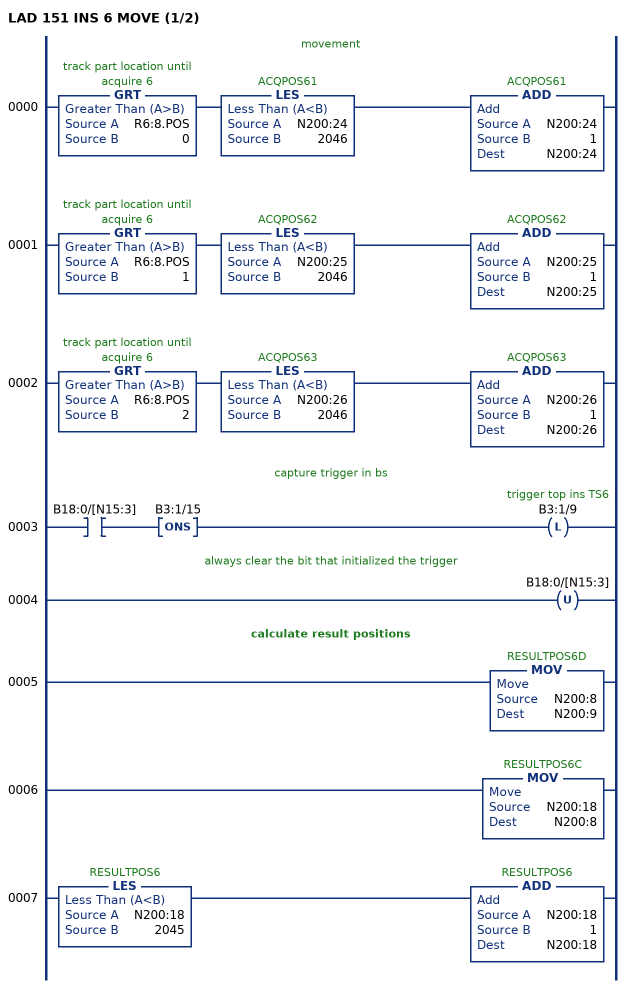
% Rung: 0 %
% movement %
SOR GRT R6:8.POS 0 LES N200:24 2046 ADD N200:24 1 N200:24 EOR
%   R6:8  "track part location until acquire 6" %
%   N200:24  ACQPOS61 %
% Rung: 1 %
SOR GRT R6:8.POS 1 LES N200:25 2046 ADD N200:25 1 N200:25 EOR
%   R6:8  "track part location until acquire 6" %
%   N200:25  ACQPOS62 %
% Rung: 2 %
SOR GRT R6:8.POS 2 LES N200:26 2046 ADD N200:26 1 N200:26 EOR
%   R6:8  "track part location until acquire 6" %
%   N200:26  ACQPOS63 %
% Rung: 3 %
% capture trigger in bs %
SOR XIC B18:0/[N15:3] ONS B3:1/15 OTL B3:1/9 EOR
%   N15:3  INS_6_TRIG_LOC %
%   B3:1/9  TS6  "trigger top ins" %
% Rung: 4 %
% always clear the bit that initialized the trigger %
SOR OTU B18:0/[N15:3] EOR
%   N15:3  INS_6_TRIG_LOC %
% Rung: 5 %
% TITLE: calculate result positions %
SOR MOV N200:8 N200:9 EOR
%   N200:8  RESULTPOS6C %
%   N200:9  RESULTPOS6D %
% Rung: 6 %
SOR MOV N200:18 N200:8 EOR
%   N200:18  RESULTPOS6 %
%   N200:8  RESULTPOS6C %
% Rung: 7 %
SOR LES N200:18 2045 ADD N200:18 1 N200:18 EOR
%   N200:18  RESULTPOS6 %

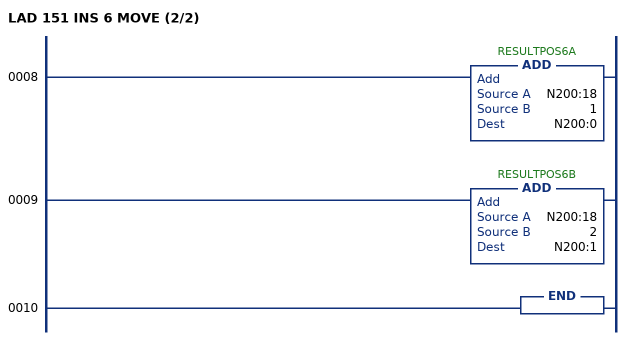
% Rung: 8 %
SOR ADD N200:18 1 N200:0 EOR
%   N200:18  RESULTPOS6 %
%   N200:0  RESULTPOS6A %
% Rung: 9 %
SOR ADD N200:18 2 N200:1 EOR
%   N200:18  RESULTPOS6 %
%   N200:1  RESULTPOS6B %
% Rung: 10 %
SOR END EOR

LADDER 160 "INS 5 TIME"
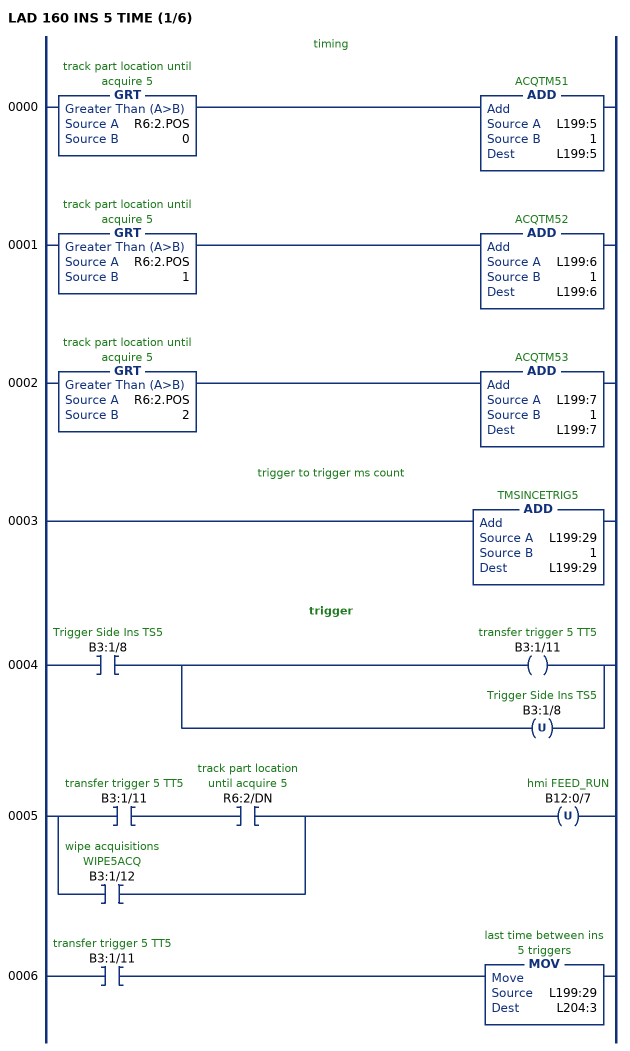
% Rung: 0 %
% timing %
SOR GRT R6:2.POS 0 ADD L199:5 1 L199:5 EOR
%   R6:2  "track part location until acquire 5" %
%   L199:5  ACQTM51 %
% Rung: 1 %
SOR GRT R6:2.POS 1 ADD L199:6 1 L199:6 EOR
%   R6:2  "track part location until acquire 5" %
%   L199:6  ACQTM52 %
% Rung: 2 %
SOR GRT R6:2.POS 2 ADD L199:7 1 L199:7 EOR
%   R6:2  "track part location until acquire 5" %
%   L199:7  ACQTM53 %
% Rung: 3 %
% trigger to trigger ms count %
SOR ADD L199:29 1 L199:29 EOR
%   L199:29  TMSINCETRIG5 %
% Rung: 4 %
% TITLE: trigger %
SOR XIC B3:1/8 BST OTE B3:1/11 NXB OTU B3:1/8 BND EOR
%   B3:1/8  TS5  "Trigger Side Ins" %
%   B3:1/11  TT5  "transfer trigger 5" %
% Rung: 5 %
SOR BST XIC B3:1/11 XIC R6:2/DN NXB XIC B3:1/12 BND OTU B12:0/7 EOR
%   B3:1/11  TT5  "transfer trigger 5" %
%   R6:2  "track part location until acquire 5" %
%   B3:1/12  WIPE5ACQ  "wipe acquisitions" %
%   B12:0/7  FEED_RUN  "hmi" %
% Rung: 6 %
SOR XIC B3:1/11 MOV L199:29 L204:3 EOR
%   B3:1/11  TT5  "transfer trigger 5" %
%   L199:29  TMSINCETRIG5 %
%   L204:3  "last time between ins 5 triggers" %

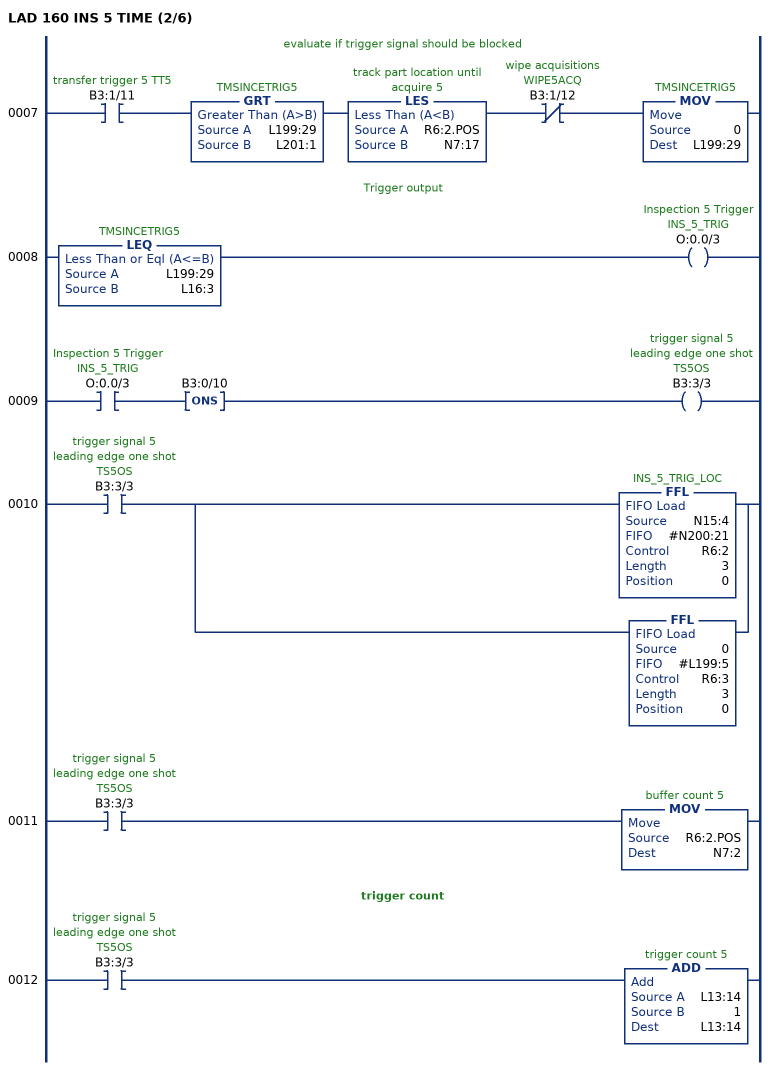
% Rung: 7 %
% evaluate if trigger signal should be blocked %
SOR XIC B3:1/11 GRT L199:29 L201:1 LES R6:2.POS N7:17 XIO B3:1/12 MOV 0 L199:29 EOR
%   B3:1/11  TT5  "transfer trigger 5" %
%   L199:29  TMSINCETRIG5 %
%   L201:1  CAM_5_MIN_CY %
%   R6:2  "track part location until acquire 5" %
%   B3:1/12  WIPE5ACQ  "wipe acquisitions" %
% Rung: 8 %
% Trigger output %
SOR LEQ L199:29 L16:3 OTE O:0.0/3 EOR
%   L199:29  TMSINCETRIG5 %
%   L16:3  CAM_5_TRIG_TIME %
%   O:0.0/3  INS_5_TRIG  "Inspection 5 Trigger" %
% Rung: 9 %
SOR XIC O:0.0/3 ONS B3:0/10 OTE B3:3/3 EOR
%   O:0.0/3  INS_5_TRIG  "Inspection 5 Trigger" %
%   B3:3/3  TS5OS  "trigger signal 5 leading edge one shot" %
% Rung: 10 %
SOR XIC B3:3/3 BST FFL N15:4 #N200:21 R6:2 3 0 NXB FFL 0 #L199:5 R6:3 3 0 BND EOR
%   B3:3/3  TS5OS  "trigger signal 5 leading edge one shot" %
%   N15:4  INS_5_TRIG_LOC %
%   N200:21  ACQPOS51 %
%   R6:2  "track part location until acquire 5" %
%   L199:5  ACQTM51 %
%   R6:3  "track acquire time 5" %
% Rung: 11 %
SOR XIC B3:3/3 MOV R6:2.POS N7:2 EOR
%   B3:3/3  TS5OS  "trigger signal 5 leading edge one shot" %
%   R6:2  "track part location until acquire 5" %
%   N7:2  "buffer count 5" %
% Rung: 12 %
% TITLE: trigger count %
SOR XIC B3:3/3 ADD L13:14 1 L13:14 EOR
%   B3:3/3  TS5OS  "trigger signal 5 leading edge one shot" %
%   L13:14  "trigger count 5" %

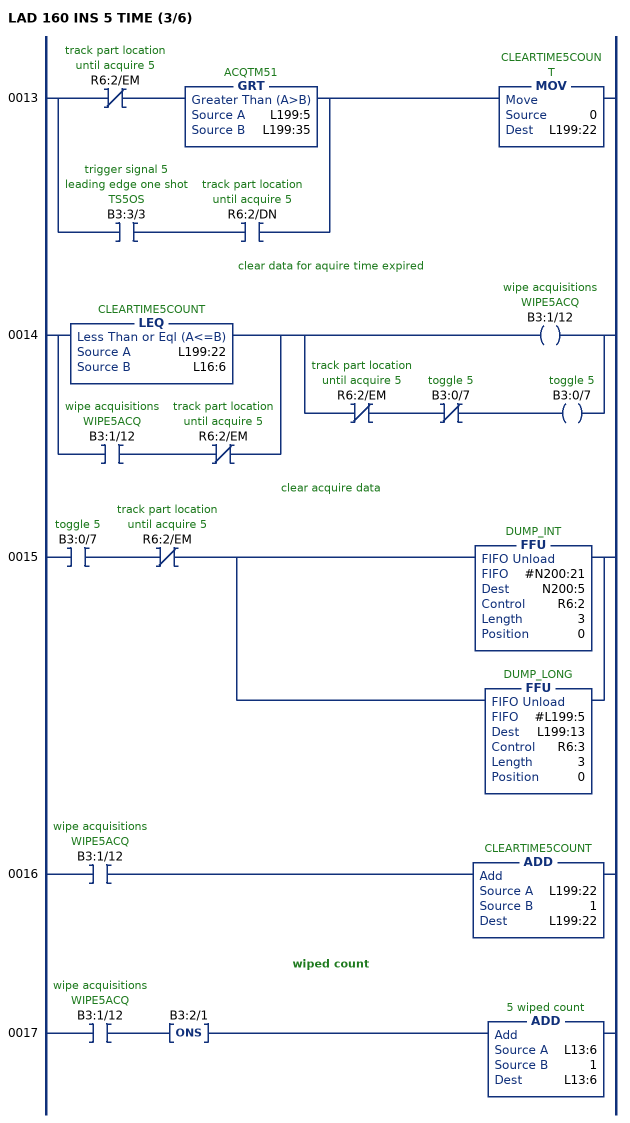
% Rung: 13 %
SOR BST XIO R6:2/EM GRT L199:5 L199:35 NXB XIC B3:3/3 XIC R6:2/DN BND MOV 0 L199:22 EOR
%   R6:2  "track part location until acquire 5" %
%   L199:5  ACQTM51 %
%   L199:35  MAXACQTM5 %
%   B3:3/3  TS5OS  "trigger signal 5 leading edge one shot" %
%   L199:22  CLEARTIME5COUNT %
% Rung: 14 %
% clear data for aquire time expired %
SOR BST LEQ L199:22 L16:6 NXB XIC B3:1/12 XIO R6:2/EM BND BST OTE B3:1/12 NXB XIO R6:2/EM XIO B3:0/7 OTE B3:0/7 BND EOR
%   L199:22  CLEARTIME5COUNT %
%   L16:6  CLEARTIME5 %
%   B3:1/12  WIPE5ACQ  "wipe acquisitions" %
%   R6:2  "track part location until acquire 5" %
%   B3:0/7  "toggle 5" %
% Rung: 15 %
% clear acquire data %
SOR XIC B3:0/7 XIO R6:2/EM BST FFU #N200:21 N200:5 R6:2 3 0 NXB FFU #L199:5 L199:13 R6:3 3 0 BND EOR
%   B3:0/7  "toggle 5" %
%   R6:2  "track part location until acquire 5" %
%   N200:21  ACQPOS51 %
%   N200:5  DUMP_INT %
%   L199:5  ACQTM51 %
%   L199:13  DUMP_LONG %
%   R6:3  "track acquire time 5" %
% Rung: 16 %
SOR XIC B3:1/12 ADD L199:22 1 L199:22 EOR
%   B3:1/12  WIPE5ACQ  "wipe acquisitions" %
%   L199:22  CLEARTIME5COUNT %
% Rung: 17 %
% TITLE: wiped count %
SOR XIC B3:1/12 ONS B3:2/1 ADD L13:6 1 L13:6 EOR
%   B3:1/12  WIPE5ACQ  "wipe acquisitions" %
%   L13:6  "5 wiped count" %

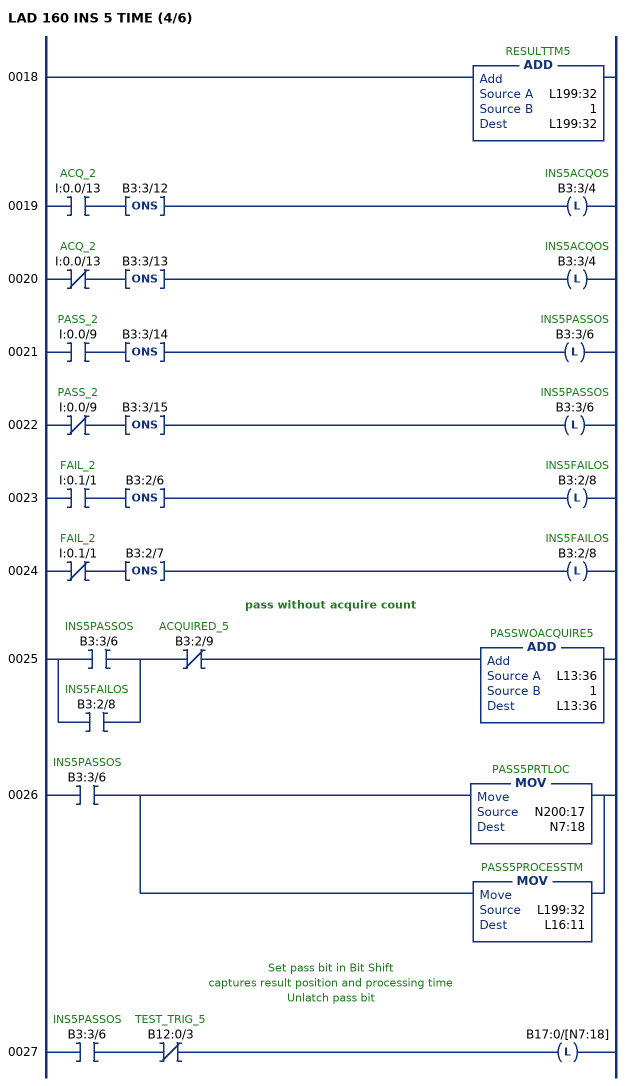
% Rung: 18 %
SOR ADD L199:32 1 L199:32 EOR
%   L199:32  RESULTTM5 %
% Rung: 19 %
SOR XIC I:0.0/13 ONS B3:3/12 OTL B3:3/4 EOR
%   I:0.0/13  ACQ_2 %
%   B3:3/4  INS5ACQOS %
% Rung: 20 %
SOR XIO I:0.0/13 ONS B3:3/13 OTL B3:3/4 EOR
%   I:0.0/13  ACQ_2 %
%   B3:3/4  INS5ACQOS %
% Rung: 21 %
SOR XIC I:0.0/9 ONS B3:3/14 OTL B3:3/6 EOR
%   I:0.0/9  PASS_2 %
%   B3:3/6  INS5PASSOS %
% Rung: 22 %
SOR XIO I:0.0/9 ONS B3:3/15 OTL B3:3/6 EOR
%   I:0.0/9  PASS_2 %
%   B3:3/6  INS5PASSOS %
% Rung: 23 %
SOR XIC I:0.1/1 ONS B3:2/6 OTL B3:2/8 EOR
%   I:0.1/1  FAIL_2 %
%   B3:2/8  INS5FAILOS %
% Rung: 24 %
SOR XIO I:0.1/1 ONS B3:2/7 OTL B3:2/8 EOR
%   I:0.1/1  FAIL_2 %
%   B3:2/8  INS5FAILOS %
% Rung: 25 %
% TITLE: pass without acquire count %
SOR BST XIC B3:3/6 NXB XIC B3:2/8 BND XIO B3:2/9 ADD L13:36 1 L13:36 EOR
%   B3:3/6  INS5PASSOS %
%   B3:2/8  INS5FAILOS %
%   B3:2/9  ACQUIRED_5 %
%   L13:36  PASSWOACQUIRE5 %
% Rung: 26 %
SOR XIC B3:3/6 BST MOV N200:17 N7:18 NXB MOV L199:32 L16:11 BND EOR
%   B3:3/6  INS5PASSOS %
%   N200:17  RESULTPOS5 %
%   N7:18  PASS5PRTLOC %
%   L199:32  RESULTTM5 %
%   L16:11  PASS5PROCESSTM %
% Rung: 27 %
% Set pass bit in Bit Shift
% captures result position and processing time
% Unlatch pass bit %
SOR XIC B3:3/6 XIO B12:0/3 OTL B17:0/[N7:18] EOR
%   B3:3/6  INS5PASSOS %
%   B12:0/3  TEST_TRIG_5 %
%   N7:18  PASS5PRTLOC %

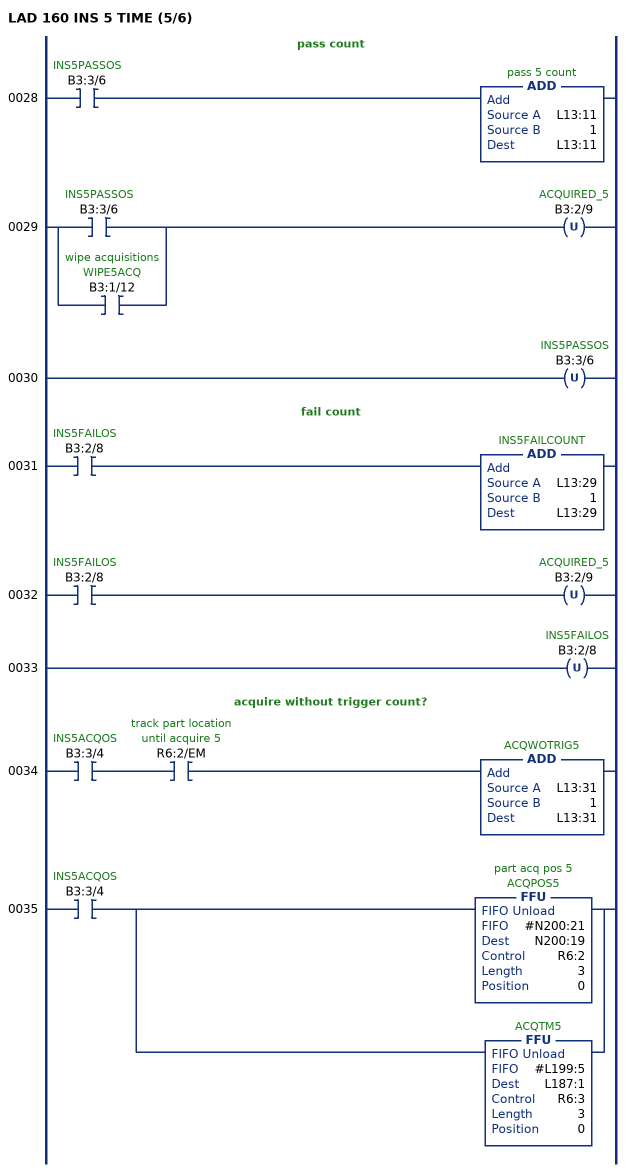
% Rung: 28 %
% TITLE: pass count %
SOR XIC B3:3/6 ADD L13:11 1 L13:11 EOR
%   B3:3/6  INS5PASSOS %
%   L13:11  "pass 5 count" %
% Rung: 29 %
SOR BST XIC B3:3/6 NXB XIC B3:1/12 BND OTU B3:2/9 EOR
%   B3:3/6  INS5PASSOS %
%   B3:1/12  WIPE5ACQ  "wipe acquisitions" %
%   B3:2/9  ACQUIRED_5 %
% Rung: 30 %
SOR OTU B3:3/6 EOR
%   B3:3/6  INS5PASSOS %
% Rung: 31 %
% TITLE: fail count %
SOR XIC B3:2/8 ADD L13:29 1 L13:29 EOR
%   B3:2/8  INS5FAILOS %
%   L13:29  INS5FAILCOUNT %
% Rung: 32 %
SOR XIC B3:2/8 OTU B3:2/9 EOR
%   B3:2/8  INS5FAILOS %
%   B3:2/9  ACQUIRED_5 %
% Rung: 33 %
SOR OTU B3:2/8 EOR
%   B3:2/8  INS5FAILOS %
% Rung: 34 %
% TITLE: acquire without trigger count? %
SOR XIC B3:3/4 XIC R6:2/EM ADD L13:31 1 L13:31 EOR
%   B3:3/4  INS5ACQOS %
%   R6:2  "track part location until acquire 5" %
%   L13:31  ACQWOTRIG5 %
% Rung: 35 %
SOR XIC B3:3/4 BST FFU #N200:21 N200:19 R6:2 3 0 NXB FFU #L199:5 L187:1 R6:3 3 0 BND EOR
%   B3:3/4  INS5ACQOS %
%   N200:21  ACQPOS51 %
%   N200:19  ACQPOS5  "part acq pos 5" %
%   R6:2  "track part location until acquire 5" %
%   L199:5  ACQTM51 %
%   L187:1  ACQTM5 %
%   R6:3  "track acquire time 5" %

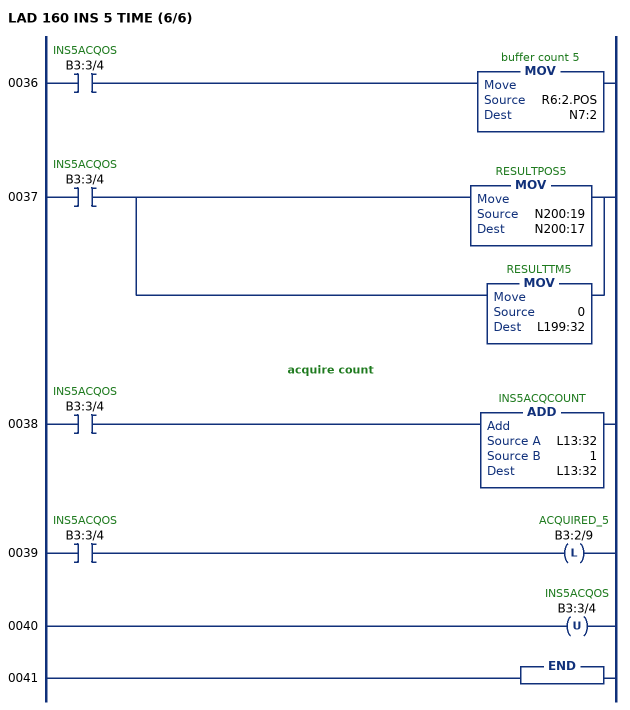
% Rung: 36 %
SOR XIC B3:3/4 MOV R6:2.POS N7:2 EOR
%   B3:3/4  INS5ACQOS %
%   R6:2  "track part location until acquire 5" %
%   N7:2  "buffer count 5" %
% Rung: 37 %
SOR XIC B3:3/4 BST MOV N200:19 N200:17 NXB MOV 0 L199:32 BND EOR
%   B3:3/4  INS5ACQOS %
%   N200:19  ACQPOS5  "part acq pos 5" %
%   N200:17  RESULTPOS5 %
%   L199:32  RESULTTM5 %
% Rung: 38 %
% TITLE: acquire count %
SOR XIC B3:3/4 ADD L13:32 1 L13:32 EOR
%   B3:3/4  INS5ACQOS %
%   L13:32  INS5ACQCOUNT %
% Rung: 39 %
SOR XIC B3:3/4 OTL B3:2/9 EOR
%   B3:3/4  INS5ACQOS %
%   B3:2/9  ACQUIRED_5 %
% Rung: 40 %
SOR OTU B3:3/4 EOR
%   B3:3/4  INS5ACQOS %
% Rung: 41 %
SOR END EOR

LADDER 161 "INS 6 TIME"
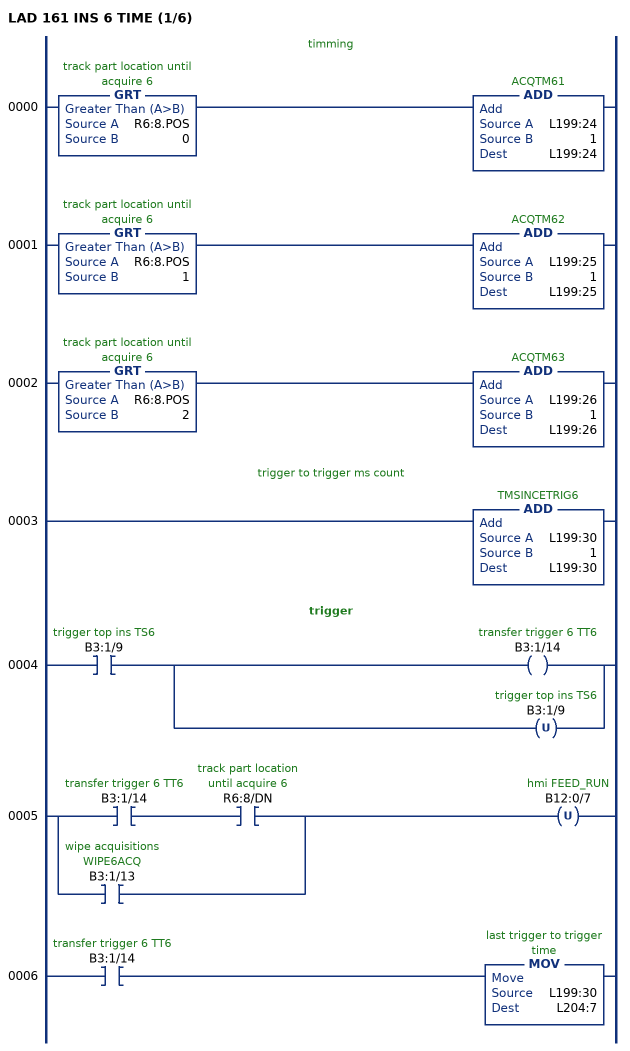
% Rung: 0 %
% timming %
SOR GRT R6:8.POS 0 ADD L199:24 1 L199:24 EOR
%   R6:8  "track part location until acquire 6" %
%   L199:24  ACQTM61 %
% Rung: 1 %
SOR GRT R6:8.POS 1 ADD L199:25 1 L199:25 EOR
%   R6:8  "track part location until acquire 6" %
%   L199:25  ACQTM62 %
% Rung: 2 %
SOR GRT R6:8.POS 2 ADD L199:26 1 L199:26 EOR
%   R6:8  "track part location until acquire 6" %
%   L199:26  ACQTM63 %
% Rung: 3 %
% trigger to trigger ms count %
SOR ADD L199:30 1 L199:30 EOR
%   L199:30  TMSINCETRIG6 %
% Rung: 4 %
% TITLE: trigger %
SOR XIC B3:1/9 BST OTE B3:1/14 NXB OTU B3:1/9 BND EOR
%   B3:1/9  TS6  "trigger top ins" %
%   B3:1/14  TT6  "transfer trigger 6" %
% Rung: 5 %
SOR BST XIC B3:1/14 XIC R6:8/DN NXB XIC B3:1/13 BND OTU B12:0/7 EOR
%   B3:1/14  TT6  "transfer trigger 6" %
%   R6:8  "track part location until acquire 6" %
%   B3:1/13  WIPE6ACQ  "wipe acquisitions" %
%   B12:0/7  FEED_RUN  "hmi" %
% Rung: 6 %
SOR XIC B3:1/14 MOV L199:30 L204:7 EOR
%   B3:1/14  TT6  "transfer trigger 6" %
%   L199:30  TMSINCETRIG6 %
%   L204:7  "last trigger to trigger time" %

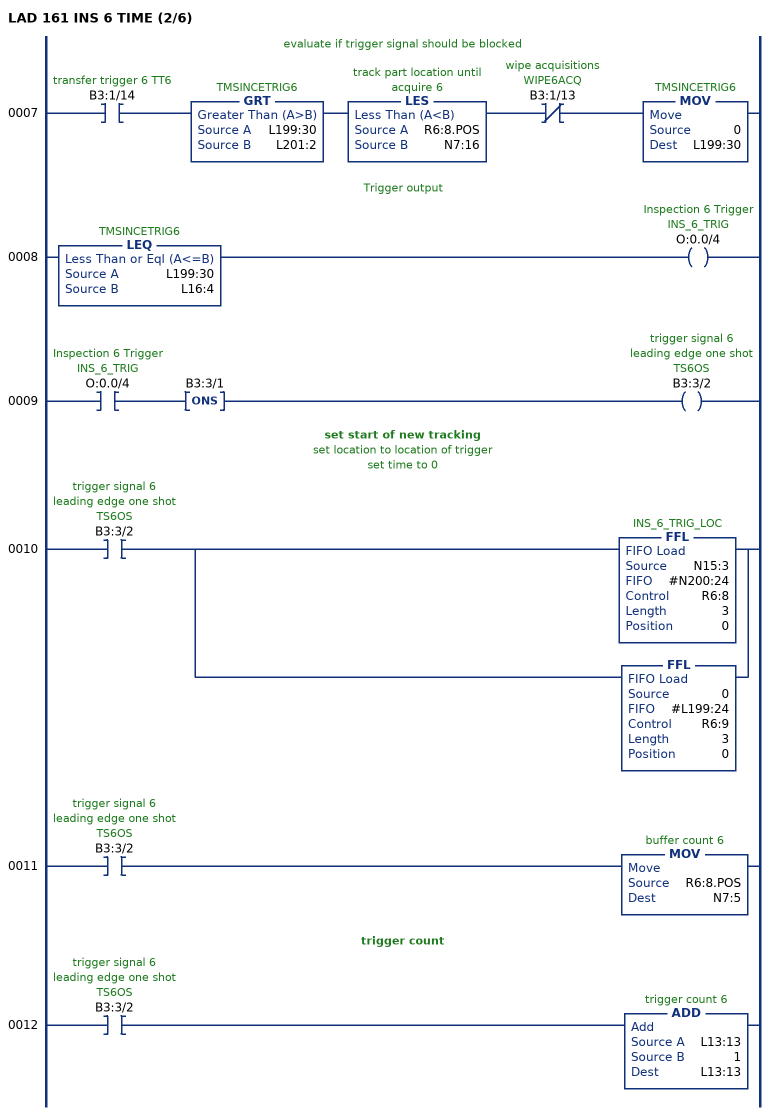
% Rung: 7 %
% evaluate if trigger signal should be blocked %
SOR XIC B3:1/14 GRT L199:30 L201:2 LES R6:8.POS N7:16 XIO B3:1/13 MOV 0 L199:30 EOR
%   B3:1/14  TT6  "transfer trigger 6" %
%   L199:30  TMSINCETRIG6 %
%   L201:2  CAM_6_MIN_CY %
%   R6:8  "track part location until acquire 6" %
%   B3:1/13  WIPE6ACQ  "wipe acquisitions" %
% Rung: 8 %
% Trigger output %
SOR LEQ L199:30 L16:4 OTE O:0.0/4 EOR
%   L199:30  TMSINCETRIG6 %
%   L16:4  CAM_6_TRIG_TIME %
%   O:0.0/4  INS_6_TRIG  "Inspection 6 Trigger" %
% Rung: 9 %
SOR XIC O:0.0/4 ONS B3:3/1 OTE B3:3/2 EOR
%   O:0.0/4  INS_6_TRIG  "Inspection 6 Trigger" %
%   B3:3/2  TS6OS  "trigger signal 6 leading edge one shot" %
% Rung: 10 %
% TITLE: set start of new tracking %
% set location to location of trigger
% set time to 0 %
SOR XIC B3:3/2 BST FFL N15:3 #N200:24 R6:8 3 0 NXB FFL 0 #L199:24 R6:9 3 0 BND EOR
%   B3:3/2  TS6OS  "trigger signal 6 leading edge one shot" %
%   N15:3  INS_6_TRIG_LOC %
%   N200:24  ACQPOS61 %
%   R6:8  "track part location until acquire 6" %
%   L199:24  ACQTM61 %
%   R6:9  "track acquire time 6" %
% Rung: 11 %
SOR XIC B3:3/2 MOV R6:8.POS N7:5 EOR
%   B3:3/2  TS6OS  "trigger signal 6 leading edge one shot" %
%   R6:8  "track part location until acquire 6" %
%   N7:5  "buffer count 6" %
% Rung: 12 %
% TITLE: trigger count %
SOR XIC B3:3/2 ADD L13:13 1 L13:13 EOR
%   B3:3/2  TS6OS  "trigger signal 6 leading edge one shot" %
%   L13:13  "trigger count 6" %

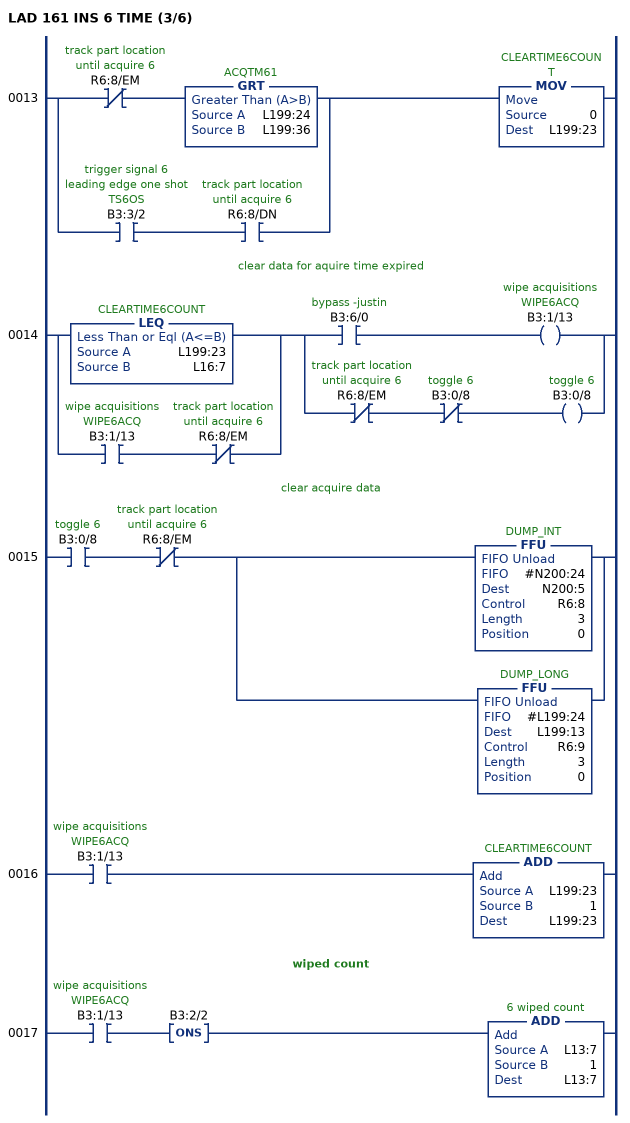
% Rung: 13 %
SOR BST XIO R6:8/EM GRT L199:24 L199:36 NXB XIC B3:3/2 XIC R6:8/DN BND MOV 0 L199:23 EOR
%   R6:8  "track part location until acquire 6" %
%   L199:24  ACQTM61 %
%   L199:36  MAXACQTM6 %
%   B3:3/2  TS6OS  "trigger signal 6 leading edge one shot" %
%   L199:23  CLEARTIME6COUNT %
% Rung: 14 %
% clear data for aquire time expired %
SOR BST LEQ L199:23 L16:7 NXB XIC B3:1/13 XIO R6:8/EM BND BST XIC B3:6/0 OTE B3:1/13 NXB XIO R6:8/EM XIO B3:0/8 OTE B3:0/8 BND EOR
%   L199:23  CLEARTIME6COUNT %
%   L16:7  CLEARTIME6 %
%   B3:1/13  WIPE6ACQ  "wipe acquisitions" %
%   R6:8  "track part location until acquire 6" %
%   B3:6/0  "bypass -justin" %
%   B3:0/8  "toggle 6" %
% Rung: 15 %
% clear acquire data %
SOR XIC B3:0/8 XIO R6:8/EM BST FFU #N200:24 N200:5 R6:8 3 0 NXB FFU #L199:24 L199:13 R6:9 3 0 BND EOR
%   B3:0/8  "toggle 6" %
%   R6:8  "track part location until acquire 6" %
%   N200:24  ACQPOS61 %
%   N200:5  DUMP_INT %
%   L199:24  ACQTM61 %
%   L199:13  DUMP_LONG %
%   R6:9  "track acquire time 6" %
% Rung: 16 %
SOR XIC B3:1/13 ADD L199:23 1 L199:23 EOR
%   B3:1/13  WIPE6ACQ  "wipe acquisitions" %
%   L199:23  CLEARTIME6COUNT %
% Rung: 17 %
% TITLE: wiped count %
SOR XIC B3:1/13 ONS B3:2/2 ADD L13:7 1 L13:7 EOR
%   B3:1/13  WIPE6ACQ  "wipe acquisitions" %
%   L13:7  "6 wiped count" %

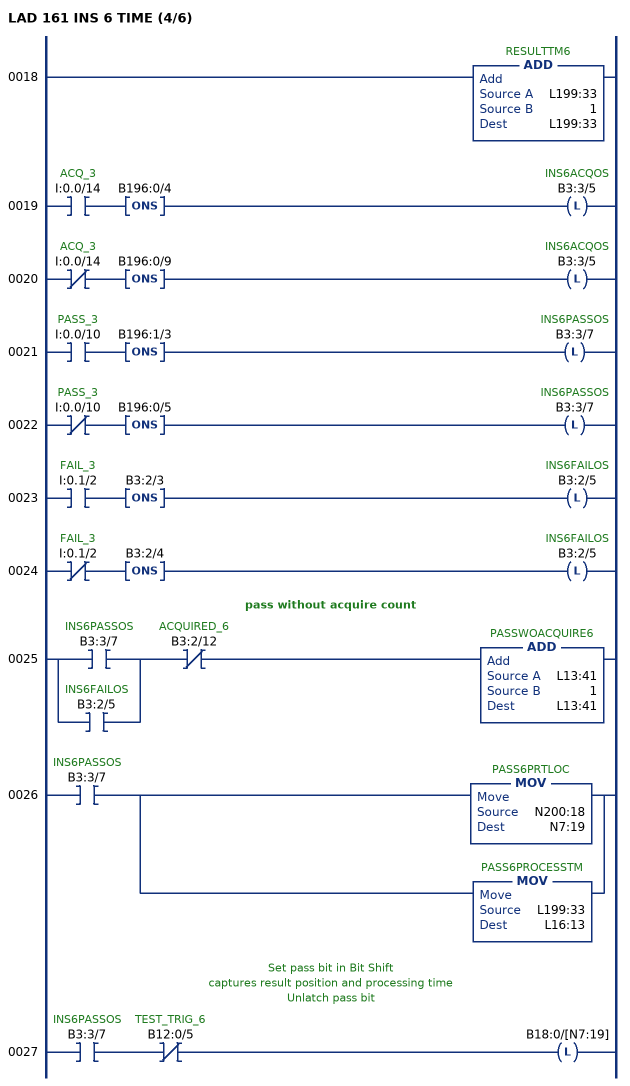
% Rung: 18 %
SOR ADD L199:33 1 L199:33 EOR
%   L199:33  RESULTTM6 %
% Rung: 19 %
SOR XIC I:0.0/14 ONS B196:0/4 OTL B3:3/5 EOR
%   I:0.0/14  ACQ_3 %
%   B3:3/5  INS6ACQOS %
% Rung: 20 %
SOR XIO I:0.0/14 ONS B196:0/9 OTL B3:3/5 EOR
%   I:0.0/14  ACQ_3 %
%   B3:3/5  INS6ACQOS %
% Rung: 21 %
SOR XIC I:0.0/10 ONS B196:1/3 OTL B3:3/7 EOR
%   I:0.0/10  PASS_3 %
%   B3:3/7  INS6PASSOS %
% Rung: 22 %
SOR XIO I:0.0/10 ONS B196:0/5 OTL B3:3/7 EOR
%   I:0.0/10  PASS_3 %
%   B3:3/7  INS6PASSOS %
% Rung: 23 %
SOR XIC I:0.1/2 ONS B3:2/3 OTL B3:2/5 EOR
%   I:0.1/2  FAIL_3 %
%   B3:2/5  INS6FAILOS %
% Rung: 24 %
SOR XIO I:0.1/2 ONS B3:2/4 OTL B3:2/5 EOR
%   I:0.1/2  FAIL_3 %
%   B3:2/5  INS6FAILOS %
% Rung: 25 %
% TITLE: pass without acquire count %
SOR BST XIC B3:3/7 NXB XIC B3:2/5 BND XIO B3:2/12 ADD L13:41 1 L13:41 EOR
%   B3:3/7  INS6PASSOS %
%   B3:2/5  INS6FAILOS %
%   B3:2/12  ACQUIRED_6 %
%   L13:41  PASSWOACQUIRE6 %
% Rung: 26 %
SOR XIC B3:3/7 BST MOV N200:18 N7:19 NXB MOV L199:33 L16:13 BND EOR
%   B3:3/7  INS6PASSOS %
%   N200:18  RESULTPOS6 %
%   N7:19  PASS6PRTLOC %
%   L199:33  RESULTTM6 %
%   L16:13  PASS6PROCESSTM %
% Rung: 27 %
% Set pass bit in Bit Shift
% captures result position and processing time
% Unlatch pass bit %
SOR XIC B3:3/7 XIO B12:0/5 OTL B18:0/[N7:19] EOR
%   B3:3/7  INS6PASSOS %
%   B12:0/5  TEST_TRIG_6 %
%   N7:19  PASS6PRTLOC %

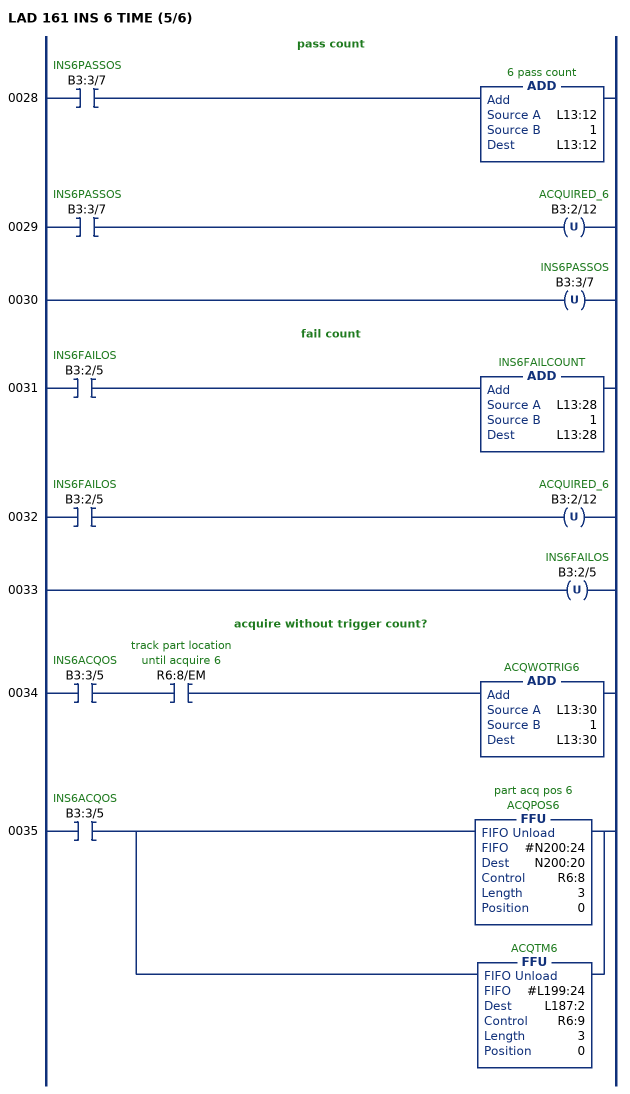
% Rung: 28 %
% TITLE: pass count %
SOR XIC B3:3/7 ADD L13:12 1 L13:12 EOR
%   B3:3/7  INS6PASSOS %
%   L13:12  "6 pass count" %
% Rung: 29 %
SOR XIC B3:3/7 OTU B3:2/12 EOR
%   B3:3/7  INS6PASSOS %
%   B3:2/12  ACQUIRED_6 %
% Rung: 30 %
SOR OTU B3:3/7 EOR
%   B3:3/7  INS6PASSOS %
% Rung: 31 %
% TITLE: fail count %
SOR XIC B3:2/5 ADD L13:28 1 L13:28 EOR
%   B3:2/5  INS6FAILOS %
%   L13:28  INS6FAILCOUNT %
% Rung: 32 %
SOR XIC B3:2/5 OTU B3:2/12 EOR
%   B3:2/5  INS6FAILOS %
%   B3:2/12  ACQUIRED_6 %
% Rung: 33 %
SOR OTU B3:2/5 EOR
%   B3:2/5  INS6FAILOS %
% Rung: 34 %
% TITLE: acquire without trigger count? %
SOR XIC B3:3/5 XIC R6:8/EM ADD L13:30 1 L13:30 EOR
%   B3:3/5  INS6ACQOS %
%   R6:8  "track part location until acquire 6" %
%   L13:30  ACQWOTRIG6 %
% Rung: 35 %
SOR XIC B3:3/5 BST FFU #N200:24 N200:20 R6:8 3 0 NXB FFU #L199:24 L187:2 R6:9 3 0 BND EOR
%   B3:3/5  INS6ACQOS %
%   N200:24  ACQPOS61 %
%   N200:20  ACQPOS6  "part acq pos 6" %
%   R6:8  "track part location until acquire 6" %
%   L199:24  ACQTM61 %
%   L187:2  ACQTM6 %
%   R6:9  "track acquire time 6" %

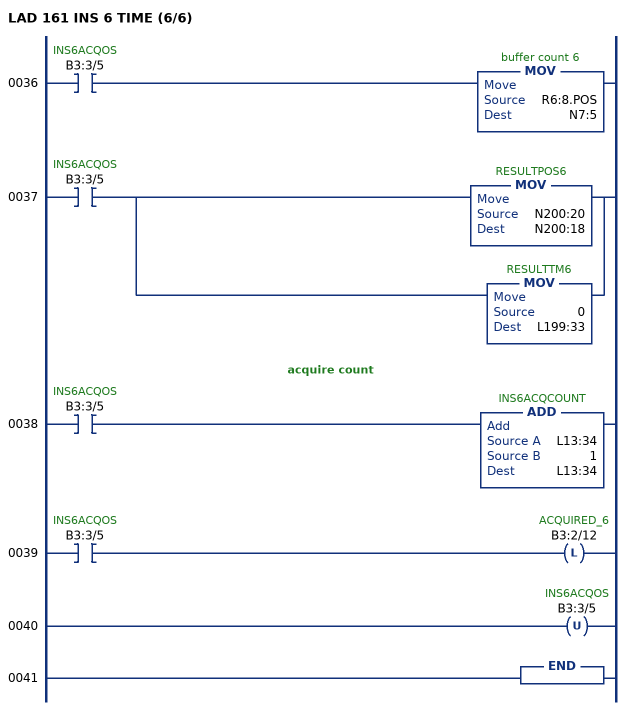
% Rung: 36 %
SOR XIC B3:3/5 MOV R6:8.POS N7:5 EOR
%   B3:3/5  INS6ACQOS %
%   R6:8  "track part location until acquire 6" %
%   N7:5  "buffer count 6" %
% Rung: 37 %
SOR XIC B3:3/5 BST MOV N200:20 N200:18 NXB MOV 0 L199:33 BND EOR
%   B3:3/5  INS6ACQOS %
%   N200:20  ACQPOS6  "part acq pos 6" %
%   N200:18  RESULTPOS6 %
%   L199:33  RESULTTM6 %
% Rung: 38 %
% TITLE: acquire count %
SOR XIC B3:3/5 ADD L13:34 1 L13:34 EOR
%   B3:3/5  INS6ACQOS %
%   L13:34  INS6ACQCOUNT %
% Rung: 39 %
SOR XIC B3:3/5 OTL B3:2/12 EOR
%   B3:3/5  INS6ACQOS %
%   B3:2/12  ACQUIRED_6 %
% Rung: 40 %
SOR OTU B3:3/5 EOR
%   B3:3/5  INS6ACQOS %
% Rung: 41 %
SOR END EOR

LADDER 170 "PASS BLOW"
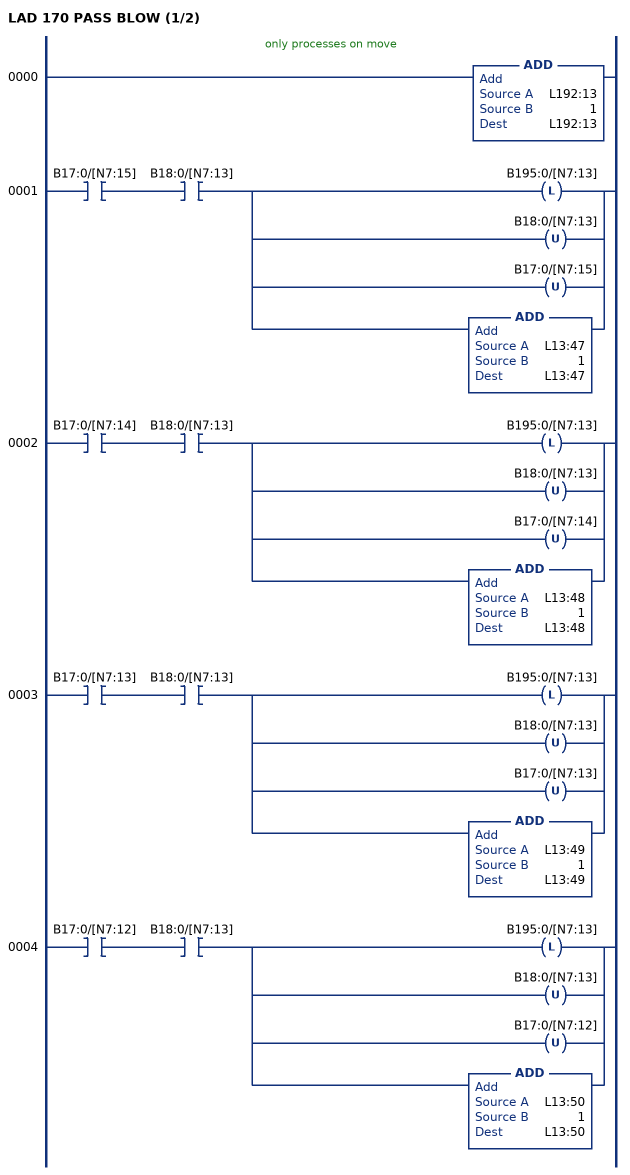
% Rung: 0 %
% only processes on move %
SOR ADD L192:13 1 L192:13 EOR
% Rung: 1 %
SOR XIC B17:0/[N7:15] XIC B18:0/[N7:13] BST OTL B195:0/[N7:13] NXB OTU B18:0/[N7:13] NXB OTU B17:0/[N7:15] NXB ADD L13:47 1 L13:47 BND EOR
%   N7:15  OS5 %
%   N7:13  OS3 %
% Rung: 2 %
SOR XIC B17:0/[N7:14] XIC B18:0/[N7:13] BST OTL B195:0/[N7:13] NXB OTU B18:0/[N7:13] NXB OTU B17:0/[N7:14] NXB ADD L13:48 1 L13:48 BND EOR
%   N7:14  OS4 %
%   N7:13  OS3 %
% Rung: 3 %
SOR XIC B17:0/[N7:13] XIC B18:0/[N7:13] BST OTL B195:0/[N7:13] NXB OTU B18:0/[N7:13] NXB OTU B17:0/[N7:13] NXB ADD L13:49 1 L13:49 BND EOR
%   N7:13  OS3 %
% Rung: 4 %
SOR XIC B17:0/[N7:12] XIC B18:0/[N7:13] BST OTL B195:0/[N7:13] NXB OTU B18:0/[N7:13] NXB OTU B17:0/[N7:12] NXB ADD L13:50 1 L13:50 BND EOR
%   N7:12  OS2 %
%   N7:13  OS3 %

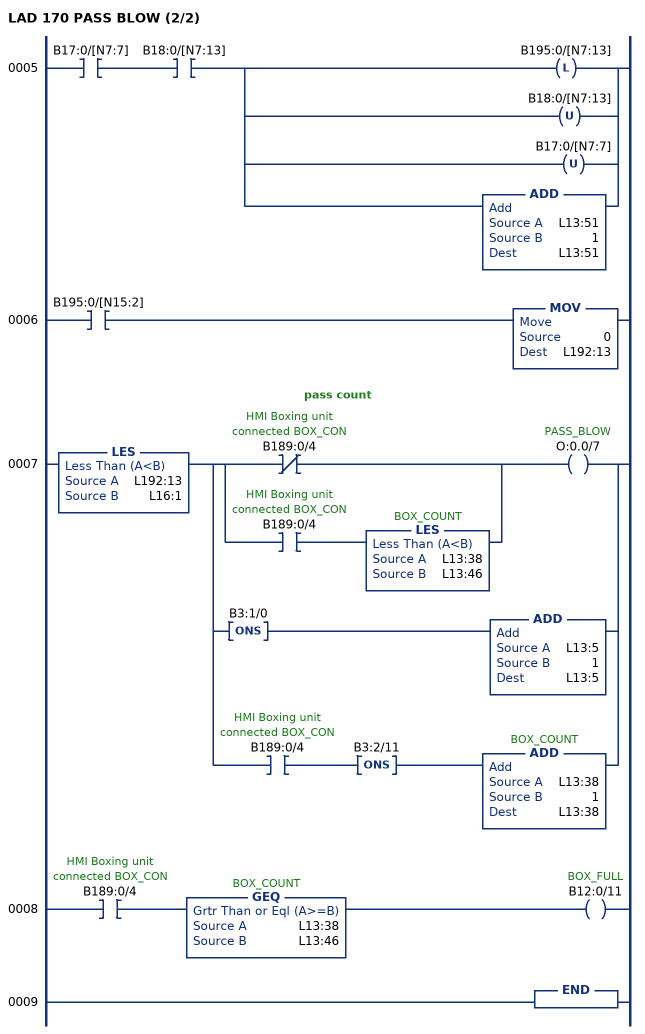
% Rung: 5 %
SOR XIC B17:0/[N7:7] XIC B18:0/[N7:13] BST OTL B195:0/[N7:13] NXB OTU B18:0/[N7:13] NXB OTU B17:0/[N7:7] NXB ADD L13:51 1 L13:51 BND EOR
%   N7:7  OS1 %
%   N7:13  OS3 %
% Rung: 6 %
SOR XIC B195:0/[N15:2] MOV 0 L192:13 EOR
%   N15:2  BLOW_PT %
% Rung: 7 %
% TITLE: pass count %
SOR LES L192:13 L16:1 BST BST XIO B189:0/4 NXB XIC B189:0/4 LES L13:38 L13:46 BND OTE O:0.0/7 NXB ONS B3:1/0 ADD L13:5 1 L13:5 NXB XIC B189:0/4 ONS B3:2/11 ADD L13:38 1 L13:38 BND EOR
%   L16:1  BLOW_TIME %
%   B189:0/4  BOX_CON  "HMI Boxing unit connected" %
%   L13:38  BOX_COUNT %
%   L13:46  BOX_LIMIT  "box count setpoint" %
%   O:0.0/7  PASS_BLOW %
% Rung: 8 %
SOR XIC B189:0/4 GEQ L13:38 L13:46 OTE B12:0/11 EOR
%   B189:0/4  BOX_CON  "HMI Boxing unit connected" %
%   L13:38  BOX_COUNT %
%   L13:46  BOX_LIMIT  "box count setpoint" %
%   B12:0/11  BOX_FULL %
% Rung: 9 %
SOR END EOR

LADDER 180 "RATE"
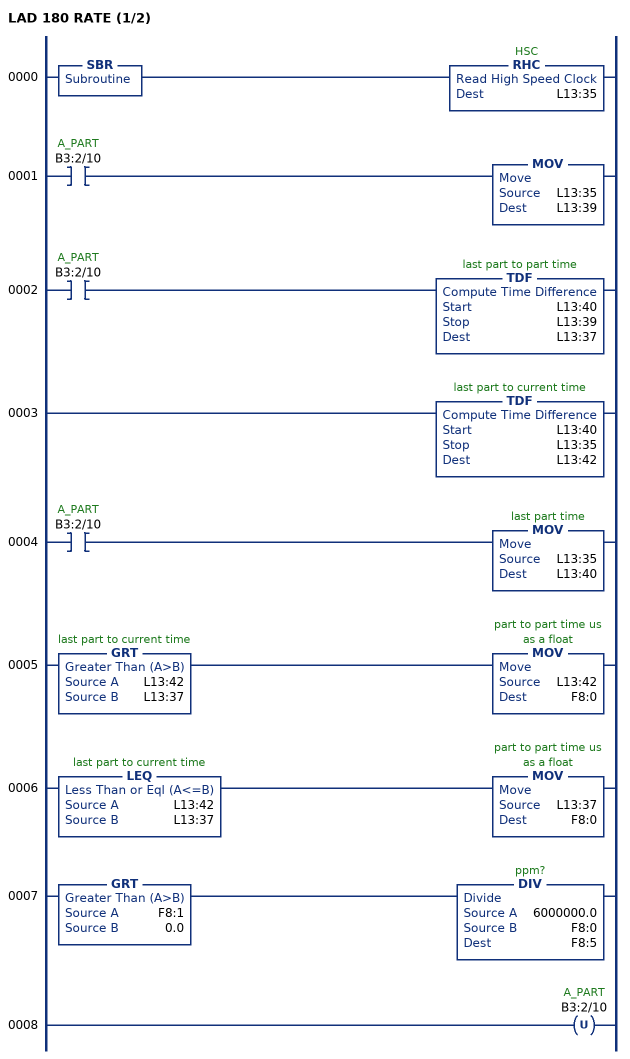
% Rung: 0 %
SOR SBR RHC L13:35 EOR
%   L13:35  HSC %
% Rung: 1 %
SOR XIC B3:2/10 MOV L13:35 L13:39 EOR
%   B3:2/10  A_PART %
%   L13:35  HSC %
% Rung: 2 %
SOR XIC B3:2/10 TDF L13:40 L13:39 L13:37 EOR
%   B3:2/10  A_PART %
%   L13:40  "last part time" %
%   L13:37  "last part to part time" %
% Rung: 3 %
SOR TDF L13:40 L13:35 L13:42 EOR
%   L13:40  "last part time" %
%   L13:35  HSC %
%   L13:42  "last part to current time" %
% Rung: 4 %
SOR XIC B3:2/10 MOV L13:35 L13:40 EOR
%   B3:2/10  A_PART %
%   L13:35  HSC %
%   L13:40  "last part time" %
% Rung: 5 %
SOR GRT L13:42 L13:37 MOV L13:42 F8:0 EOR
%   L13:42  "last part to current time" %
%   L13:37  "last part to part time" %
%   F8:0  "part to part time us as a float" %
% Rung: 6 %
SOR LEQ L13:42 L13:37 MOV L13:37 F8:0 EOR
%   L13:42  "last part to current time" %
%   L13:37  "last part to part time" %
%   F8:0  "part to part time us as a float" %
% Rung: 7 %
SOR GRT F8:1 0.0 DIV 6000000.0 F8:0 F8:5 EOR
%   F8:0  "part to part time us as a float" %
%   F8:5  "ppm?" %
% Rung: 8 %
SOR OTU B3:2/10 EOR
%   B3:2/10  A_PART %

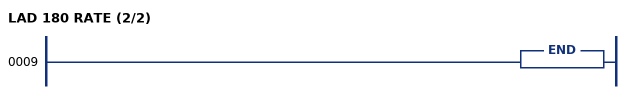
% Rung: 9 %
SOR END EOR

OTHER DOCUMENTED ADDRESSES
  B3:8/1  "bypass extra trigger camera 2"
  B3:8/2  "bypass extra trigger camera 3"
  B3:8/3  "bypass extra trigger camera 4"
  B3:8/6  "a bypass bit"
  B3:8/7  "a bypass bit"
  B3:8/12  "start bottom top camera responce"
  B3:8/13  "extra blow signal for testing"
  B3:8/15  "start side camera responce"
  B3:9/2  "one shot"
  B3:9/4  "start top camera responce"
  B3:9/6  "C1D"
  B3:9/7  "C1t"
  B3:9/8  "C2D"
  B3:9/9  "C2t"
  B3:9/14  "input from hmi to reset count"
  B3:10/0  "bypass part too close"
  B3:10/2  "One Shot"
  B3:10/3  "One Shot"
  B3:10/4  "changing Box chute door operation"
  B3:10/5  "one shot"
  B3:10/6  "excessive data output time"
  B3:10/9  "one shot"
  B3:10/10  "one shot"
  B3:10/11  "bottom part present trailling edge"
  B3:10/13  "one shot"
  B3:10/14  "Dont use"
  B3:10/15  "Reserved For Shift Registers"
  B3:11/0  "bypass unused portion of code"
  B3:11/1  "bypass"
  B3:11/2  "Enable encoder belt movement simulation when testing"
  B3:11/3  "Block blow signals while changing box"
  B3:11/4  "one shot"
  B3:11/6  "one shot"
  B3:11/7  "one shot"
  B3:11/8  "one shot"
  B3:11/11  "one shot"
  B3:11/12  "one shot"
  B3:11/15  "one shot"
  B3:12/0  "one shot"
  B3:12/1  "one shot"
  B3:12/2  "Command 2 Oneshot"
  B3:12/3  "Command 2 Active"
  B3:12/4  "Command3 Oneshot"
  B3:12/5  "Command 3 Active"
  B3:12/6  "Inspection Command Counter"
  B3:12/7  "Command 4 Active"
  B3:12/8  "Command 4 Oneshot"
  B3:12/14  "flip flop bit"
  B3:13/5  "bypass"
  B3:13/6  "Off"
  B3:13/7  "On"
  B3:13/8  "On"
  B3:13/9  "Off"
  B3:13/10  "On"
  B3:13/11  "Off"
  B3:13/12  "Test Trigger to laser Spacing"
  B3:13/15  "Test Signals"
  B3:17/12  "Always Off"
  B9:0/0  "Trigger Insert Position"
  B9:0/1  "bottom of top conveyor part transfer location"
  B9:0/[N7:0]  "Side Camera Trigger Posistion"
  B9:0/[N7:2]  "Mask Start Position"
  B9:0/[N7:6]  "Blow Off Position"
  B9:0/[N7:20]  "part present bit shift load position"
  B9:0/[N7:48]  "Top Camera Trigger Posistion"
  B9:0/[N16:0]  "Trigger Position"
  B9:0/[N17:8]  "part from bottom belt present at top belt optic position"
  B10:0/0  "Pass Insert Position"
  B10:0/[N7:2]  "Pass Bit Position"
  B10:0/[N7:4]  "Pass Insert Position"
  B10:0/[N7:5]  "Pass Start Position"
  B10:0/[N7:6]  "Pass Position"
  B10:0/[N16:4]  "Pass Insert Position"
  B10:0/[N16:6]  "Pass Position"
  B11:0/0  "Trigger Insert Position"
  B11:0/[N7:8]  "Fail Bit Position"
  B11:0/[N16:0]  "Trigger Position"
  B12:1/0  "Conveyor Start Oneshot"
  B12:1/1  "Feed Start Oneshot"
  B12:1/2  "Conveyor Stop Oneshot"
  B12:1/3  "Feed Stop Oneshot"
  B12:1/5  "Conveyor Start Oneshot"
  B12:10  BULK_PACK
  B14:0/0  "Bottom Pass Insert"
  B14:0/4  "Bottom Pass Insert Position"
  B14:0/[N13:14]  "Start Laser Pass"
  B14:0/[N16:4]  "Pass Insert Position"
  B14:0/[N16:6]  "Pass Position"
  B15:0  "Alarm Bits"
  B18:1/1  "bottom pass one shot transfer"
  B18:3/2  "Part Present Oneshot"
  B18:3/3  "Part Present Oneshot"
  B18:5/11  "Transfer bottom pass result from end of bottom conveyor"
  B18:10/15  "Reserved For Shift Registers"
  B18:142  "fack camerea pass signal"
  B22:0  "Transfer Shift Register"
  B22:0/0  "load top conveyor bitshift from bottom cammera pass."
  B22:0/[N17:8]  "bottom good part at top optic position"
  B23:0/[N7:0]  "Bottom Pass Output"
  B185:0/0  "bypass"
  B185:0/1  "bypass"
  B185:0/9  "result time 1 okay"
  B185:0/11  "test fail out"
  B185:0/12  "enable"
  B185:0/13  "enable"
  B185:1/0  "enable"
  B185:1/3  "enable"
  B185:1/7  "enable"
  B191:1/0  "Part measured wider then the limit set in the optic test"
  B191:1/1  "part to part spacing smaller then the set minimum value"
  B191:1/2  "Boxing conveyor backed up"
  B191:2/0  "bottom to top alignment"
  B196:0/13  "waiting for result"
  B196:0/14  "acquire before result os"
  B196:0/15  "enable count"
  B196:1/5  "switch me to EN_1"
  B196:1/9  "Enable alignment Signal"
  B196:1/11  "enable"
  B196:1/12  "enable"
  B196:1/15  "transfer trigger for position alignment logical one shot"
  B196:2/0  "enable"
  B196:2/2  "enable"
  B196:2/8  "enable count"
  B196:2/9  "time out 1"
  B196:2/10  "Reset bad head fault"
  B196:4/0  "test trigger signal 1"
  B196:4/4  "real part within distance of virtual part"
  B196:4/15  "pass in bit shift"
  F8:13  "error top"
  F8:15  "error bottom"
  F8:20  "bot belt speed average in pulses per second"
  F8:26  "Part bits loaded into BitShift"
  F8:28  "momentary rate in ppm"
  F8:29  "Count of signals passed to the blow valve"
  F8:31  "Count of off alignment between top and bottom ALIGN_FAILS"
  F8:34  "count of blow signals"
  F8:35  "rate difference"
  F8:38  "averaged rate"
  F8:40  "absoloute difference top"
  F8:41  "absoloute difference bottom"
  F8:42  "Total fail and missed count CAM_NON_PASS"
  F8:43  "change in part rate as %"
  F8:44  "difference as a ratio of the total"
  F8:45  "TOO_CLOSE_BOT"
  F8:46  "TOO_WIDE_BOT"
  F8:48  "transfer"
  F8:49  "TOO_CLOSE_TOP"
  F8:51  "TOO_WIDE_TOP"
  F8:52  "OPTO_FAILS"
  F8:53  "optic fail count top camera TOP_OPT_FAIL_CT"
  F8:54  "optic fail count bot camera BOT_OPT_FAIL_CT"
  F19:4  "Conveyor Input Blip Counter"
  F188:1  "HMI Recerk speed input"
  F188:2  "HMI input for feed wheel speed"
  F188:3  "HMI input for feeder speed"
  F188:4  "HMI input for hopper speed"
  F192:0  "temp"
  F205:0  "feed wheel"
  F205:1  "feed bowl"
  F205:2  "hopper"
  HSC:0.3/6  "Underflow interrupt"
  HSC:0.3/7  "Overflow interrupt"
  HSC:1.3/6  "Underflow interrupt"
  HSC:1.3/7  "Overflow interrupt"
  I:0.0/0  "Encoder Signal "A""
  I:0.0/1  "Encoder Signal "B""
  I:0.0/4  "Encoder Signal "A""
  I:0.0/5  "Encoder Signal "B""
  I:0.0/11  PASS_4
  I:0.0/15  ACQ_4
  I:0.1/3  FAIL_4
  I:0.2/3  "Packaging Conveyor full"
  I:0.2/4  "Packaging Conveyor Box in Position"
  I:0.4  "Spare Analog Input 1"
  I:0.5  "Spare Analog Input 2"
  I:0.6  "Spare Analog Input 3"
  I:2.0/1  REAR_ESTOP
  I:2.0/8  "front door signal"
  I:2.0/9  "rear door signal"
  I:2.0/10  "Maintenance Key Switch"
  I:2.0/12  "input from customer Packager Concluded"
  L23:1  MPCE_ON
  L23:19  TOP_OPT_FAIL_CT
  L23:34  AIR_PRESSURE_FAULT
  L183:2  "simulated part width"
  L187:5  "pass transfer out signals"
  L187:6  "NoErr transfer out signals"
  L187:7  "ins 1 trigger count"
  L190:0  "count of bottom optic width fails"
  L190:1  "count of gap fails"
  L190:2  "I1 blocked triggers"
  L190:4  "count of parts rejected because acquire time ran out"
  L190:5  "count of parts that received a pass signal but previously failed 1"
  L190:6  "count of result signals received with no part present 1"
  L190:7  "count of results received after maximim time reached"
  L190:8  "pass count"
  L190:9  "fail count"
  L190:10  "acquisition count"
  L190:11  "acquisition without result count"
  L190:12  "count of parts results that time out"
  L190:27  "optic alignment pass signal"
  L190:28  "optic alignment fail signal"
  L190:31  "something wrong, can't happen"
  L190:32  "Crazy wrong, can't happen"
  L201:5  "ms since trig 1 is initialized"
  L201:10  "movement from virtual (pos, add)"
  L204:13  "This optic signal time"
  L204:14  "Last optic signal time"
  L204:15  "time between optic signals"
  N10:1  "old ConveyorStatus"
  N10:2  "PowerOn"
  N10:3  "Local Mode On BypassBoxingPLC"
  N10:4  "Boxing Connected Signal"
  N10:5  "BoxJamSignal"
  N10:6  "WaittingOnBoxSig"
  N10:7  "ConveyorFullSig"
  N10:8  "MachineFaultSig"
  N10:9  "Counter Sensor Fault"
  N10:11  "Feeder Track Sensor Blocked"
  N10:12  "Air Pressure Fault"
  N13:0  "Part Inspecting"
  N13:4  "Completed Counter"
  N13:5  "Trigger Position Counter"
  N13:6  "BlowOff Start Counter"
  N13:7  "BlowOff Stop Counter"
  N13:8  "Inspection Command Counter"
  N13:9  "Complete Counter"
  N13:10  "Pass Signal Counter"
  N13:11  "Solenoid Signal Counter"
  N13:12  "Hold Pass Counter"
  N13:13  "Hold Pass Length"
  N16:1  "Bottom Inspection Offset For Tracking"
  N16:3  "Bit Shift Preset"
  N17:5  "Parts In Tube Counter"
  N17:6  "Parts In Tube Limit"
  N17:9  "Bot to Top Transfer Position"
  N17:12  "Trigger to laser Counter"
  N197:1  "maximim acquire time 1"
  N197:5  "Feeder Speed Output Setting"
  N197:10  "pulse distance to keep blow on then turn off feed"
  N197:11  "speed in pps"
  N197:12  "seconds of ontime"
  N197:20/0  "Deformed Head Blowoff Bit to TOP PLC"
  O:0.0/1  "spare"
  O:0.0/5  INS_4_TRIG
  O:0.0/6  "spare"
  O:0.0/11  "Spare"
  O:0.5  "spare"
  O:3.0/0  "Ready-Run signal to Boxer? Always on unless fault?"
  O:3.0/2  "Customers pecies counting done signal (Change Box?)"
  O:3.0/6  RED_LT  "Red Light"
  O:3.0/7  "Spare"
  O:3.0/8  "spare"
  PFILE:6  "check for part jams"
  PFILE:10  "Bottom belt HSC"
  PFILE:12  "Top belt HSC"
  Q2:55  END_OF_MAIN
  Q5:94  END_OF_BELTS
  R6:5.POS  "Empty Fifo"
  R21:0  "Trigger Shift Register"
  T4:7  "Boxing conveyor full error delay"
  T4:9  "optio hold holds minimum optic time to 16ms"
  T4:11  "belt stop delay timer"
  T4:12  "Hopper On Delay"
  T4:17  "Stopped Time Out Timer"
  T4:23  "SETUP TIMER"
  T4:24  "bot cam responce timmer 2"
  T4:25  "box in posistion pulse stretcher timer"
  T4:27  "Timer to allow parts to pass through shoot"
  T4:28  "Timer to allow shoot door to close"
  T4:29  "Part Rate Timer"
  T4:30  "Hopper Off Delay"
  T4:32  "Deformed Head Blowoff Timer"
  T20:0  "Trigger On Time"
  U:5  "conveyor"
  U:9  "slow data"
  U:11  "transfered data calcuations from the high speed section"
  U:28  "faults"
  U:29  "speed"
  U:30  "count"
  U:31  "rate calc"
  U:32  "boxer"
  U:33  "bulk pack"
  U:34  "customer boxing unit signals"
  U:35  "cleanup"
  U:95  "HMI interface"
  U:120  "simulate part injection"
  U:121  "bot optic"
  U:130  "transfer to top"
  U:140  "top optic"

COMMENTS NOT ATTACHED TO A CURRENT RUNG
  N17:8: ****************************************************************************************************************
    I can not find anywhere in the program where the "Test Spacing From Pickup to Trigger is activated indicating to me that this entire function must not be doing anything in this program at this time.
    ****************************************************************************************************************
  T20:2: The timer used to verify that the part that triggered the top laser optic has passed the bottom camer. needs to be count
  T20:2.ACC: This rung is starting a timer that should be activated directly before the laser optic part presense sensor on the top conveyer and should cause the top optic to be ignored if the bottom camera system didn't pass. however other arrangements must be made if the bottom camera isn't going to be used as is the case with a nut inspection.
  B22:0/0: ***********************
     Bottom Part Syncronizing Logic
    ***********************
    
    This is the point at the bottom of the top conveyor where the part jumps from the bottom conveyor.  This system will then track the part through the top system to the point of the laser optic in order to verify that the part in question has passed the bottom inspection.  I believe that we NEED to include FAILING inspections to eliminate the possibility of a out of position part from passing. LW 072010
  C5:4: tempory counting to verify pass part count with boxing part count.
  N7:25: 1050
  B23:0/0: Yet another bit shift load with data in the part position indicating that there was a bottom system part pass as well as a top system part present at this location.
    
    verified works w/bypassed 071910 and unbypassed 072010
  I:0.0/8: special rung for testing. This rung can simulate a pass signal. It will not be timed correctly.
  F8:13: *************************
    Loads Side Camera Passing data into a bit shift
    *************************
    
    loads passing data bit into passing data bit shift register at the part present cl.
  B3:7/9: ************************************
     The next 3 rungs appear to do nothing
    ***********************************
  B11:0/0: load part present bit shit with one shot data from the part present sensor
  N7:45: not fully functional because of part overlap but measurems the camera responce time when part inspections are not overlaping
  B3:6/1: ***********************
    Part Width and  Location
    ***********************
    
    Calculates the position of parts on the top belt by measureing the part width by calculating the number of belt movement pulses that occure when the optic is blocked and then devides that in half and add that to the optic location in the part presnet bit shift when the top optic is cleared.
  B3:6/0: make a bit come on indicating that a part that passed the bottom camera is within  range when crossing the top camera.
  B9:0/[N7:47]: Remove any part present signals outside of expected location
  O:0.0/3: **************
    Side Camera Trigger
    *************
  B9:0/[N7:50]: Remove any part present signals outside of expected location
  B3:4/14: *****
    Convertion of the optic signal to something stable
    *****
  F19:0: Counter inside of a high speed counter interrupt counts the number of Bit Shifts that need to be processed in order to move the logic with the parts on the conveyor.
  F8:14: **************
    Bottom Top Camera Trigger
    *************
    
    Trigger Bottom Top Camera
  B3:6/8: ********************************************************************************************************************************
    Box count reached
    Redo all of boxing;
    1. handle box done, change, box not moving, no new box
    2. everything else is situational, i.e. box removed, box not present
    add bulk pack rutine that just stops bowl and doesn't change box.
    ********************************************************************************************************************************
  N10:4: test if boxing is connected
  T4:27: Time to clear shoot
  T4:28: Time to close shoot door
  B3:11/3: After initial delay allow blow two start functioning
  B3:6/9: Detect fault condition no box present on conveyor
  RUNG000150-000041: transfer tracked part positon from trigger/acquire to the acquire/result
    capture acquire time
    reset process time
  RUNG000150-000039: Grab trigger/acquire position
    Grab acquire time
  RUNG000150-000038: acquire code
  RUNG000150-000035: fail count
  RUNG000150-000032: pass count
  RUNG000150-000025: pass code / Set pass bit in Bit Shift
    captures result position and processing time
    Unlatch pass bit
  RUNG000150-000018: pass, fail and acquire inputs
  RUNG000150-000016: wiped count
  RUNG000150-000014: clear data for time
  RUNG000150-000013: clear data for aquire time expired
  RUNG000150-000012: wipe stored part data if acq time expires
  RUNG000150-000011: trigger count
  L14:5: on when ok to run, rear off turns both off
  L14:2: off when ok to run
  L14:3: off when ok to run
  L14:8: on when ok for run
  N7:76: removed relieance on trigger signal
  N197:20/0: Passes deformed head blowoff command to TOP PLC where solenoid output is located.
  N7:47: ***********************************************************************************************************************************************************
    From side
    ***********************************************************************************************************************************************************
    
    removed relieance on trigger signal
  N7:50: ***********************************************************************************************************************************************************
    From top
    ***********************************************************************************************************************************************************
    
    removed relieance on trigger signal
  B3:10/1: prevents momentary signals from box present sensor from tripping the logic for box not present
    
    This is in responce to a problem created by the sensor occasionally turning on as if no box was in its path when there is a box present.
  B3:6/2: IF PROCESSING FAULT OCURES AT COUNTER SENSOR; CLEAR THE BELT OF PASSING DATA
  L14:36: ****************  nEEDS fIXING  **********************
  L14:23: ****************  nEEDS fIXING  **********************
  RUNG000010-000018: Remove any part present signals outside of expected location
  RUNG000010-000014: ****
                      Zeros out the non passing part count when one passes
    ****
  RUNG000125-000007: Trigger output
  RUNG000125-000011: trigger count
  RUNG000125-000012: wipe stored part data if acq time expires
  RUNG000125-000013: clear data for aquire time expired
  RUNG000125-000014: clear data for time
  RUNG000125-000016: wiped count
  RUNG000125-000018: pass, fail and acquire inputs
  RUNG000125-000025: pass code / Set pass bit in Bit Shift
    captures result position and processing time
    Unlatch pass bit
  RUNG000125-000026: Grab trigger/acquire position
    Grab acquire time
  RUNG000125-000027: transfer tracked part positon from trigger/acquire to the acquire/result
    capture acquire time
    reset process time
  RUNG000125-000029: Set pass bit in Bit Shift
    captures result position and processing time
    Unlatch pass bit
  N7:46: Remove any part present signals outside of expected location

REVISION NOTES
  13: updated count reset
  14: added io moduals
  15: multiple steps toward new hmi integration
  21: test

DATA TABLE (non-zero values as saved)
DATA B3
% B3:0 % 0X9021 0X0050 0X4090 0XA100 0X0306 0X2000 0X02C1 0X0020 0X4007 0X0000
% B3:10 % 0X2041 0X0846 0X2000 0X0000
DATA T4
% .PRE .ACC %
% T4:0 % 300 304
% T4:1 % 150 0
% T4:2 % 32765 0
% T4:3 % 32765 0
% T4:4 % 32765 0
% T4:5 % 150 150
% T4:6 % 5555 3363
% T4:7 % 10 0
% T4:8 % 300 0
% T4:9 % 30 0
% T4:10 % 35 0
% T4:12 % 50 0
% T4:13 % 222 0
% T4:14 % 222 0
% T4:15 % 180 0
% T4:16 % 222 0
% T4:17 % 300 0
% T4:18 % 8 0
% T4:19 % 6 0
% T4:20 % 10 0
% T4:21 % 100 0
% T4:22 % 20 0
% T4:23 % 900 0
% T4:24 % 1000 0
% T4:25 % 250 250
% T4:26 % 666 666
% T4:27 % 400 0
% T4:28 % 400 0
% T4:29 % 10 0
% T4:30 % 50 50
% T4:31 % 20 0
% T4:32 % 69 0
DATA R6
% .LEN .POS %
% R6:0 % 3 0
% R6:1 % 3 0
% R6:2 % 3 0
% R6:3 % 3 0
% R6:4 % 2048 0
% R6:5 % 2048 0
% R6:6 % 912 0
% R6:7 % 435 0
% R6:8 % 3 0
% R6:9 % 3 0
% R6:10 % 659 0
% R6:11 % 659 0
% R6:12 % 2048 0
DATA N7
% N7:0 % 6 1224 3 996 0 3 1 1611 92 75
% N7:10 % 1216 61 1610 1609 1608 1607 3 3 1223 1246
% N7:20 % 0 0 0 0 0 0 -403 0 0 0
% N7:50 % 1236 0 175 16 0 0 0 1464 12 0
% N7:60 % 1 32767 4012 20 31 0 0 15 30 20
% N7:70 % 0 21 23 27738 32767 0 122 0 16 0
% N7:80 % 0 6 95 0 0 0 5 500 0 0
% N7:90 % 2011 4 4 12 1 0 0 0 0 1600
% N7:100 % 123 124 1227 1228 1237 1238 0 0 0 0
% N7:110 % 0 0 0 0 0 0 0 0 400 0
% N7:120 % 25007 61 0 0 0 0 0 0 0 0
DATA F8
% F8:0 % 2767232 206.64 0.20664 5.736945e-05 17430.88
% F8:5 % 2.168232 0 0 0 206
% F8:10 % 0.0888 0.08897486 2322 101 63.26563
% F8:15 % 37.73437 4040 206 0 0
% F8:20 % 0 0.02 0 1 0
% F8:25 % 0 932781 0.222 279.6551 848597
% F8:30 % 0 170 0.03 38 852060
% F8:35 % 0 0 0 0 77
% F8:40 % 101 37.73437 0 100 1
% F8:45 % 1 2 0.21455 0 0
% F8:50 % 0 0 1 0 1
% F8:55 % 2000000 -221 0 0 0
% F8:95 % 0 0 0 492 4.92
DATA B9
% B9:130 % 0X0000 0X0000 0X0000 0X0000 0X2000 0X0000 0X0000 0X0000 0X0000 0X8000
% B9:140 % 0X2480 0X0000 0X0000 0X0000 0X0000 0X0000 0X0000 0X0000 0X0000 0X0000
% B9:160 % 0X0000 0X0000 0X0000 0X0000 0X0000 0X0000 0X2000 0X0002 0X0000 0X0000
% B9:170 % 0X0000 0X0000 0X0000 0X2000 0X0000 0X0000 0X0000 0X0000 0X0000 0X0000
% B9:180 % 0X0000 0X0000 0X0000 0X0000 0X0000 0X0002 0X0000 0X0000 0X0000 0X0000
% B9:190 % 0X0010 0X0000 0X0000 0X0000 0X0000 0X0000 0X0000 0X0000 0X0000 0X0000
% B9:200 % 0X2B64 0X2B64 0X0000 0X0010 0X0000 0X2000 0X0000 0X0000 0X0000 0X0000
% B9:220 % 0X0000 0X0000 0X0000 0X0200 0X0000 0X0000 0X0000 0X0000 0X0000 0X0020
% B9:230 % 0X0040 0X0000 0X0000 0X0000 0X0000 0X0000 0X0000 0X0000 0X0000 0X0000
DATA B11
% B11:180 % 0X0000 0X8000 0X0000 0X0000 0X0000 0X0000 0X0000 0X0000 0X0000 0X0000
% B11:240 % 0X0000 0X0000 0X0000 0X4000 0X0000 0X0000 0X0000 0X0000 0X0000 0X0000
DATA B12
% B12:0 % 0X0155 0X0000 0X0000 0X0000 0X0000 0X0000 0X0000 0X0000 0X0000 0X0000
DATA L13
% L13:0 % 308402300 308407124 4824 0 1000
% L13:5 % 112998 62 58 1162124017 1162124017
% L13:10 % 492 129583 116248 133455 133315
% L13:15 % 0 0 0 2147483647 82058
% L13:25 % 0 0 0 17099 3619
% L13:30 % 131 132 133198 220 133343
% L13:35 % -455960712 461 10364 0 -458815746
% L13:40 % -458815746 444 2859169 289169 31503
% L13:45 % 243785 100 10 4 4275450
% L13:50 % 5 5 2147483647 0 0
DATA F14
% F14:0 % 269.4403 270.2112 27 27 1343.406
% F14:5 % 9502.14 13106.4 982.98 0 0
DATA N15
% N15:0 % 6 908 1612 1224 1212 170 101 1204 1004 5555
% N15:10 % 62 620 0 0 0 0 1204 0 0 0
DATA L16
% L16:0 % 8 9 5 5 5
% L16:5 % 250 5000 5000 192 20
% L16:10 % 1256 18 2045 43 98
% L16:15 % 99 0 0 0 0
DATA B17
% B17:100 % 0X0000 0X0000 0X0000 0X0000 0X0000 0X0000 0X0800 0X0000 0X1000 0X0000
% B17:110 % 0X4000 0X0000 0X0000 0X0000 0X0000 0X0000 0X0000 0X0000 0X0000 0X0000
% B17:120 % 0X0000 0X0000 0X0000 0X0000 0X0000 0X0000 0X0000 0X2000
DATA B18
% B18:100 % 0X0000 0X0000 0X0000 0X0000 0X0000 0X0001 0X0000 0X0080 0X0000 0X8240
% B18:110 % 0X0000 0X0400 0X0000 0X0000 0X0000 0X0000 0X0040 0X0000 0X0000 0X0010
% B18:120 % 0X0000 0X0000 0X0000 0X0000 0X0000 0X0000 0X0000 0X2000
DATA L23
% L23:0 % 65535 -65536 -65536 -65536 -65536
% L23:5 % -65536 -65536 207 65535 -65536
% L23:10 % -65536 0 17 10 17
% L23:15 % 0 0 0 0 8
% L23:20 % 0 -65536 -65536 -65536 -65536
% L23:25 % -65536 20 19 20 0
% L23:30 % 0 0 -65536 -65536 -65536
% L23:35 % -65536 -65536 -65536 -65536 -65536
% L23:40 % 16270 18414 0 63266 -65536
% L23:45 % 5062 0 0 0 0
% L23:50 % 0 -65536 -65536 17 -65536
% L23:55 % 33 5079 -65536 0 0
% L23:60 % 0 -65536 -65536 -65536 0
DATA L24
% L24:0 % -65536 122 -65536 222 -65536
% L24:5 % 65535 -65536 -65536 -65536 -65536
% L24:10 % 50 27 0 1 23
% L24:15 % 1198 1030 95 18 30
% L24:20 % 30 -65536 1226 -65536 -65536
% L24:25 % 222 1236 -65536 -65536 222
% L24:30 % 1466 27 10000 -65536 55
% L24:35 % 180 -65536 180 65535 101
% L24:40 % 101 1000 -65536 -65536 10
% L24:45 % 222 192 -65536 0 -65536
% L24:50 % -999 30 10000 65535 900
DATA L42
% L42:0 % -65536 0 0 0 0
% L42:5 % 45 45 45 0 0
% L42:20 % 0 0 32766 32766 0
% L42:50 % 0 30
DATA L183
% L183:0 % 999 216325420 12 1000000000 0
% L183:5 % 103 50 39 0 0
DATA B185
% B185:0 % 0X0200 0X0001 0X0000 0X0000 0X0000 0X0000 0X0000 0X0000 0X0000 0X0000
DATA N186
% N186:0 % 100 0 0 0 0 0 0 0 0 0
DATA L187
% L187:0 % 71 23 37 0 0
% L187:5 % 1063 0 0 0 0
DATA F188
% F188:0 % 6 66 11 44 29
DATA B189
% B189:0 % 0X00E0 0X0000 0X0000 0X0000 0X0000 0X0000 0X0000 0X0000 0X0000 0X0000
DATA L190
% L190:0 % 1 5 0 0 0
% L190:30 % 0 2 0 0 0
DATA B191
% B191:0 % 0X0000 0X0001 0X0000 0X0000 0X0000 0X0000 0X0000 0X0000 0X0000 0X0000
DATA L192
% L192:0 % -455715279 -455715279 381 41 15231
% L192:5 % 100000 13700000 999 999 8
% L192:10 % 0 0 0 9865 17
% L192:15 % -455715417 -455715417 381 41 15179
% L192:20 % 180 13600000 0 0 0
DATA F193
% F193:0 % 1.00929 0.315 0.022 6 270
% F193:5 % -0.4730225 0.15 -0.07095337 272.5084 8929.011
% F193:10 % 0.011 0.195 0.165 0.337 270
% F193:15 % -0.03414917 0.15 -0.005122376 348.7363 11426.69
DATA B195
% B195:60 % 0X0000 0X0000 0X0000 0X0000 0X0000 0X0000 0X0000 0X0000 0X4000 0X19C0
% B195:70 % 0X8000 0X84B0 0X0210 0X0000 0X0000 0X0000 0X0000 0X0000 0X0000 0X0000
DATA B196
% B196:0 % 0X0814 0X9FFE 0X0005 0X0000 0X0000 0X0000 0X0000 0X0000 0X0000 0X0000
% B196:30 % 0XE800 0X9BFF 0XEBFF 0XFFDF 0XFFFF 0X0000 0X0000 0X0000 0X0000 0X0000
DATA N197
% N197:0 % 1560 150 1111 2500 2500 14417 5555 300 150 0
% N197:10 % 4000 969 4 0 0 0 0 0 0 0
% N197:30 % 15 48 0 0 0 0 0 0 0 0
DATA B198
% B198:0 % 0X0009 0X0000 0X0000 0X0000 0X0000 0X0000 0X0000 0X0000 0X0000 0X0000
DATA L199
% L199:0 % 1 5571998 134 11 3579521
% L199:5 % 0 0 0 5 174974
% L199:10 % 0 224 10256 112 0
% L199:15 % 0 0 225 278717848 518
% L199:20 % 38325 16430853 5001 5001 0
% L199:25 % 0 0 32643 999 32624
% L199:30 % 32580 251 38392 38334 111
% L199:35 % 555 555 0 0 0
DATA N200
% N200:0 % 2046 2047 2046 2047 2045 200 1008 2045 2045 2045
% N200:10 % 0 0 0 1277 189 2046 1000 2045 2045 1218
% N200:20 % 1234 0 0 0 0 0 0 0 0 0
% N200:30 % 0 0 32767 0 0 0 0 0 0 0
DATA L201
% L201:0 % 20 40 40 -3011735 44
% L201:5 % 96629277 0 0 -3010662 0
% L201:10 % 0 0 0 327 43
% L201:15 % 0 43 0 43 36830
DATA B202
% B202:0 % 0X2241 0X0000 0X0001 0X0000 0X0000 0X0000 0X0000 0X0000 0X0000 0X0000
DATA N203
% N203:0 % 115 115 116 333 334 333 444 0 445 444
% N203:10 % 555 556 555 0 0 0 0 0 0 0
DATA L204
% L204:0 % 111 101 111 1915 501
% L204:5 % 0 0 1915 222 0
% L204:10 % 0 0 0 1327077052 1327077052
% L204:15 % 1327077052 1327077052 1 0 0
% L204:20 % 0 0 33 0 0
% L204:30 % 33 0 0 0 0
DATA F205
% F205:0 % 655.32 655.32 655.32 655.32 0
